Staubli VAL3: Digtal2AnalogS.pgx

public program Digtal2AnalogS(num x_nId (dimensions=1))
  local num l_nIndexX
  local num l_nIndexY
  local num l_nNum
  local string l_sIOName
begin

  //数字量转换为模拟量

  //0 67到82
  //1 83到98
  //2 99到114
  //3 115到130
  //4 131到146


  x_nId=min(4,max(0,x_nId))
  for l_nIndexY=x_nId to x_nId
    l_nNum=0
    for l_nIndexX=0 to 15
      call IOName(67+l_nIndexX+l_nIndexY*16,l_sIOName)
      if (67+l_nIndexX+l_nIndexY*16)<135
        l_nNum=l_nNum+sel(dDio[l_sIOName]==true,1,0)*power(2,l_nIndexX)
      endIf
    endFor
    call IOName(159+l_nIndexY,l_sIOName)
    aioSet(aAio[l_sIOName],l_nNum)
    delay(0)
  endFor



























end
